% RSLogix 500 project SOLISPLC_ML1100_BAK010.RSS, saved by version 11.00.00.00 %
PROJECT "SOLISPLC"    % processor: Bul.1763 MicroLogix 1100 Series B %

PROGRAM FILES
  LAD 2   3 rungs

DATA FILES
  O0 OUTPUT  4 elements
  I1 INPUT  6 elements
  S2 STATUS  66 elements
  B3 BINARY  1 elements
  T4 TIMER  1 elements
  C5 COUNTER  1 elements
  R6 CONTROL  1 elements
  N7 INTEGER  10 elements
  F8 FLOAT  1 elements
  L9 LONG  10 elements  % long %

LADDER 2
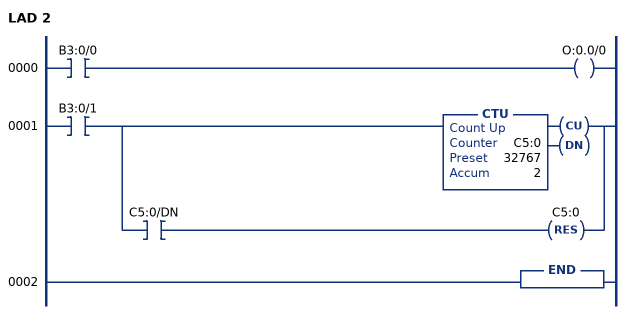
% Rung: 0 %
SOR XIC B3:0/0 OTE O:0.0/0 EOR
% Rung: 1 %
SOR XIC B3:0/1 BST CTU C5:0 32767 2 NXB XIC C5:0/DN RES C5:0 BND EOR
% Rung: 2 %
SOR END EOR

DATA TABLE (non-zero values as saved)
DATA T4
% .PRE .ACC %
% T4:0 % 10 7
DATA C5
% .PRE .ACC %
% C5:0 % 32767 2
DATA N7
% N7:0 % 32766 0 0 0 0 0 0 0 0 0
DATA L9
% L9:0 % 34298 34447 0 0 0
